TYPE
  (* Version 1.0, 2025-03-22, AK123700 *)
  position : STRUCT
    X : UINT; (* Output event qualifier *)
    Y : UINT;
    Z : UINT;
  END_STRUCT;
END_TYPE
